Yaskawa INFORM job: X2_27-28(-50,-90).JBI

/JOB
//NAME X2_27-28(-50,-90)
//POS
///NPOS 347,347,347,16,0,0
///TOOL 0
///POSTYPE PULSE
///PULSE
C00000=2348,-136985,-121477,16,96092,119
C00001=-102627,-116827,-115343,-23688,103226,44542
C00002=-115004,-86962,-92134,-24001,100691,40453
C00003=-118842,-87386,-89376,-23795,97842,39618
C00004=-120381,-87384,-88200,-23717,96741,39273
C00005=-120377,-87274,-86494,-23659,95829,39457
C00006=-120358,-87289,-86697,-23665,95942,39442
C00007=-122537,-87238,-86673,-23616,95334,38762
C00008=-120358,-87289,-86697,-23665,95942,39442
C00009=-120413,-87366,-86683,-23662,95882,39433
C00010=-120414,-83407,-84990,-23721,96794,39250
C00011=-120413,-87366,-86683,-23662,95882,39433
C00012=-118874,-87417,-87880,-23731,96972,39781
C00013=-115033,-87126,-90695,-23913,99792,40627
C00014=-115188,-84882,-91157,-24044,101067,40307
C00015=-118973,-85347,-88418,-23826,98226,39491
C00016=-120455,-85363,-87251,-23745,97137,39166
C00017=-120452,-85286,-85558,-23683,96217,39352
C00018=-120487,-85295,-85812,-23691,96347,39313
C00019=-122635,-85238,-85785,-23639,95749,38643
C00020=-120487,-85295,-85812,-23691,96347,39313
C00021=-120483,-89746,-89095,-23675,96102,39363
C00022=-120398,-93403,-88367,-23560,93986,39817
C00023=-120400,-89378,-86736,-23609,94965,39621
C00024=-120398,-93403,-88367,-23560,93986,39817
C00025=-114754,-95185,-95401,-23812,98729,40947
C00026=-113817,-96176,-94667,-23309,84492,38861
C00027=-117813,-93582,-90807,-22657,82424,37804
C00028=-119373,-92438,-89214,-22393,81636,37384
C00029=-121634,-92435,-89210,-21971,81030,36673
C00030=-120812,-92629,-89389,-22126,81259,36930
C00031=-120809,-92377,-87626,-22175,80372,37096
C00032=-120812,-92629,-89389,-22126,81259,36930
C00033=-120909,-77641,-83091,-21971,84792,36245
C00034=-120897,-73822,-81314,-21956,85603,36101
C00035=-120909,-77641,-83091,-21971,84792,36245
C00036=-115943,-80689,-88441,-22878,87717,37472
C00037=-114304,-84462,-91699,-24296,79100,50020
C00038=-117993,-82622,-88033,-23316,76858,49124
C00039=-119438,-81769,-86512,-22922,76000,48762
C00040=-121534,-81768,-86509,-22277,75434,48100
C00041=-120893,-81605,-86471,-22471,75662,48293
C00042=-120882,-79116,-84088,-22491,75491,48329
C00043=-120893,-81605,-86471,-22471,75662,48293
C00044=-120874,-97072,-87829,-23296,69089,49605
C00045=-120882,-99825,-87797,-23508,67765,49878
C00046=-120874,-97072,-87829,-23296,69089,49605
C00047=-115137,-101258,-93439,-24799,71949,51221
C00048=-121122,-106374,-107449,1374,89824,2285
C00049=-126924,-83388,-91593,24529,79629,-49999
C00050=-123244,-81641,-87969,23551,77363,-49118
C00051=-121801,-80822,-86464,23159,76497,-48761
C00052=-119718,-80838,-86473,22519,75929,-48107
C00053=-120355,-80669,-86431,22711,76157,-48297
C00054=-120355,-78205,-84050,22728,75972,-48332
C00055=-120355,-80669,-86431,22711,76157,-48297
C00056=-120389,-96242,-87887,23521,69604,-49623
C00057=-120385,-99021,-87874,23730,68282,-49899
C00058=-120389,-96242,-87887,23521,69604,-49623
C00059=-126112,-100299,-93445,25011,72503,-51215
C00060=-127424,-95125,-94496,23537,84985,-38865
C00061=-123439,-92623,-90674,22887,82890,-37821
C00062=-121881,-91514,-89094,22623,82092,-37406
C00063=-119636,-91530,-89104,22205,81483,-36703
C00064=-120453,-91715,-89278,22359,81714,-36957
C00065=-120449,-91492,-87527,22405,80819,-37124
C00066=-120453,-91715,-89278,22359,81714,-36957
C00067=-120324,-76745,-82936,22209,85198,-36262
C00068=-120328,-72933,-81149,22194,85997,-36116
C00069=-120324,-76745,-82936,22209,85198,-36262
C00070=-125282,-79685,-88237,23118,88153,-37475
C00071=-126053,-84105,-90945,24270,101400,-40334
C00072=-121317,-84665,-86997,23961,97551,-39378
C00073=-120794,-84655,-86302,23916,97014,-39294
C00074=-120791,-84616,-85408,23898,96528,-39392
C00075=-120757,-84623,-85661,23907,96658,-39353
C00076=-118619,-84583,-85646,23856,96058,-38687
C00077=-120757,-84623,-85661,23907,96658,-39353
C00078=-120851,-89642,-89189,23884,96311,-39457
C00079=-120861,-92728,-88235,23770,94318,-39863
C00080=-120850,-88708,-86596,23821,95285,-39665
C00081=-120861,-92728,-88235,23770,94318,-39863
C00082=-126087,-84100,-90943,24271,101411,-40344
C00083=-126241,-86175,-91925,24226,101032,-40481
C00084=-121422,-86671,-87791,23936,97086,-39512
C00085=-120872,-86641,-86990,23895,96491,-39430
C00086=-120871,-86598,-86346,23873,96146,-39499
C00087=-120890,-86611,-86548,23880,96260,-39483
C00088=-118722,-86577,-86536,23832,95649,-38808
C00089=-120890,-86611,-86548,23880,96260,-39483
C00090=-105063,-136064,-103329,13656,63018,-16453
C00091=-105943,-129413,-101511,13642,65401,-16501
C00092=-120836,-86689,-86535,23876,96200,-39475
C00093=-126205,-86358,-90494,24135,100129,-40655
C00094=-125851,-82973,-83923,27955,66645,-49280
C00095=-122078,-79433,-79887,26568,64829,-48204
C00096=-120742,-75548,-77663,25886,64978,-47626
C00097=-120603,-87757,-78081,27201,59519,-48941
C00098=-120577,-18765,-47570,25588,110640,-38043
C00099=-109277,-31294,-61129,11102,108845,-34159
C00100=-108190,-73941,-84391,11784,95620,-26863
C00101=-120412,-77832,-82211,23564,93525,-30308
C00102=-120295,-129804,-92806,30270,50820,-51385
C00103=-120103,-142543,-87811,36899,40276,-55620
C00104=-123719,-144899,-89705,38330,41729,-57027
C00105=-131684,-150990,-93667,41315,44633,-60156
C00106=-129569,-143343,-101170,37382,56065,-55166
C00107=-120626,-84262,-98768,23738,98439,-36527
C00108=-120626,-85138,-96217,23600,96582,-36901
C00109=-120626,-85402,-95162,23554,95859,-37045
C00110=-120626,-85402,-95166,23554,95862,-37044
C00111=-120625,-86138,-87819,24831,69352,-42364
C00112=-120624,-85351,-79999,28656,54651,-46082
C00113=-120624,-83851,-73296,29505,52526,-46737
C00114=-120624,-85502,-80901,24858,69157,-42411
C00115=-120625,-86091,-86368,23338,89997,-38197
C00116=-120623,-90747,-88263,23328,88867,-38416
C00117=-120625,-86141,-87502,23348,90617,-38076
C00118=-120625,-86117,-90396,23390,92270,-37753
C00119=-121122,-106374,-107449,1374,89824,2285
C00120=-115389,-83619,-83840,-27729,66202,49282
C00121=-119161,-80016,-79774,-26335,64406,48194
C00122=-120089,-78340,-77954,-26002,63882,47941
C00123=-118763,-53285,-67852,-25424,88543,43198
C00124=-120520,-20811,-48856,-25337,110383,38072
C00125=-120672,-56250,-71200,-24620,106276,38936
C00126=-122381,-110474,-92211,-22628,69435,43351
C00127=-117850,-143004,-85318,-49461,33775,58563
C00128=-117015,-147748,-80398,-56682,30834,62523
C00129=-116407,-166632,-89102,-63406,28902,66105
C00130=-115676,-54235,-75024,-25023,110799,39825
C00131=-118805,-64147,-80292,-27733,101935,40879
C00132=-120626,-85310,-99014,-23481,98015,36524
C00133=-120626,-86187,-96453,-23350,96148,36894
C00134=-120946,-86934,-95392,-23260,95104,36986
C00135=-120769,-87776,-95791,-23270,94982,37074
C00136=-120625,-87052,-87833,-24600,68847,42365
C00137=-120546,-85594,-79665,-28457,54282,46089
C00138=-120538,-84322,-72984,-29356,52066,46772
C00139=-120625,-86297,-80888,-24632,68687,42397
C00140=-119608,-72473,-79941,-24560,98029,43290
C00141=-120361,-60134,-73697,-25010,105724,48535
C00142=-120625,-87037,-87669,-23119,90208,38053
C00143=-120626,-87011,-90570,-23155,91868,37731
C00144=-120666,-77011,-108669,-24508,106824,34682
C00145=-69969,-70044,-127853,26190,66176,-42607
C00146=-164066,-57873,-122395,24689,68505,-41679
C00147=-164066,-57873,-122395,24689,68505,-41679
C00148=-160176,-49519,-119791,24551,119921,-39872
C00149=-160176,-63483,-121326,22850,113002,-41438
C00150=-158640,-65340,-120741,22195,111473,-41297
C00151=-158591,-68589,-120293,21868,109653,-41643
C00152=-157443,-69457,-121106,21570,109470,-41332
C00153=-156525,-70687,-121652,21280,109008,-41144
C00154=-157421,-68776,-121134,21620,109807,-41260
C00155=-165312,-86424,-128504,22962,107296,-44197
C00156=-165830,-86354,-127308,22986,106767,-44469
C00157=-165199,-83493,-126223,22948,107364,-44147
C00158=-166594,-89849,-128602,23030,106020,-44865
C00159=-164066,-57873,-122395,24689,117052,-41679
C00160=-137183,-48540,-113103,27062,110870,-33097
C00161=-133437,-50146,-110771,25387,107987,-32705
C00162=-131981,-50551,-109735,24766,106894,-32528
C00163=-131972,-53362,-109280,24521,105318,-32870
C00164=-131636,-52132,-109559,24518,105977,-32629
C00165=-130703,-53161,-109590,24138,105304,-32500
C00166=-129879,-53398,-109717,23857,105082,-32305
C00167=-131928,-52773,-109383,24556,105642,-32786
C00168=-129764,-110950,-131053,20350,81074,-33499
C00169=-129689,-122862,-131886,20674,75787,-34382
C00170=-129370,-114001,-129067,20345,78360,-33827
C00171=-129689,-122862,-131886,20674,75787,-34382
C00172=-132778,-100905,-131254,21387,86712,-33498
C00173=-143318,-75184,-130722,7426,108145,-5953
C00174=-142042,-70835,-125479,6985,107076,-5675
C00175=-141569,-69161,-123389,6821,106623,-5573
C00176=-141558,-72780,-123049,6738,104567,-5686
C00177=-141593,-72294,-123187,6761,104902,-5677
C00178=-140967,-66354,-120569,6623,106293,-5428
C00179=-141593,-72294,-123187,6761,104902,-5677
C00180=-143345,-79213,-130741,7340,106105,-6087
C00181=-143299,-74412,-130544,7434,108429,-5930
C00182=-142026,-70178,-125329,6991,107319,-5656
C00183=-141554,-68541,-123249,6826,106852,-5556
C00184=-141544,-72173,-122918,6742,104795,-5669
C00185=-141535,-71558,-123086,6755,105212,-5644
C00186=-140912,-65651,-120469,6618,106588,-5397
C00187=-141535,-71558,-123086,6755,105212,-5644
C00188=-143280,-78289,-130595,7337,106482,-6046
C00189=-143232,-73654,-130370,7428,108704,-5895
C00190=-141965,-69530,-125182,6983,107555,-5626
C00191=-141496,-67928,-123110,6817,107076,-5527
C00192=-141485,-71574,-122787,6732,105017,-5641
C00193=-141522,-70879,-122980,6762,105492,-5624
C00194=-140900,-65004,-120364,6625,106853,-5379
C00195=-141522,-70879,-122980,6762,105492,-5624
C00196=-143263,-77436,-130447,7347,106826,-6020
C00197=-97122,-37708,-107994,-29413,114613,34215
C00198=-100765,-40257,-106178,-27624,111617,33971
C00199=-102190,-41052,-105346,-26964,110463,33848
C00200=-102184,-43828,-104954,-26656,108968,34218
C00201=-102229,-43254,-105047,-26705,109274,34130
C00202=-104151,-44223,-105589,-26045,108681,33706
C00203=-102229,-43254,-105047,-26705,109274,34130
C00204=-102390,-95092,-126215,-23236,87986,35228
C00205=-102126,-106454,-127212,-23433,83236,36243
C00206=-102723,-99043,-124596,-23148,85111,35678
C00207=-102126,-106454,-127212,-23433,83236,36243
C00208=-98351,-76946,-122874,-24964,95636,34932
C00209=-98001,-57475,-123101,-17996,113820,36592
C00210=-101536,-60773,-120906,-16470,110382,36160
C00211=-102910,-63141,-119733,-15828,108317,36071
C00212=-102916,-65026,-119479,-15713,107233,36217
C00213=-102928,-64308,-119579,-15751,107645,36158
C00214=-105169,-65555,-120144,-15037,107042,35610
C00215=-102928,-64308,-119579,-15751,107645,36158
C00216=-100368,-93898,-131351,-15864,100368,37874
C00217=-97661,-87630,-128580,-16731,102276,38427
C00218=-97996,-84252,-127310,-16710,103135,38207
C00219=-97637,-87591,-128732,-16747,102389,38418
C00220=-98001,-57475,-123101,-17996,113820,36592
C00221=-99672,-7498,-88471,-25376,120102,35641
C00222=-102088,-13346,-89114,-23936,117260,35660
C00223=-103047,-14853,-89113,-23458,116364,35598
C00224=-103070,-15280,-89318,-23419,116275,35613
C00225=-103053,-14956,-89343,-23464,116445,35580
C00226=-111428,-26181,-98637,-10737,112296,30408
C00227=-102060,-12538,-89166,-24052,117675,35572
C00228=-99645,-6651,-88487,-25511,120511,35544
C00229=-110953,-13508,-91662,-10573,109125,-24437
C00230=-110055,-18058,-91129,-10746,106581,-23991
C00231=-118115,-24092,-94041,1176,104714,-22608
C00232=-109847,-18561,-90498,-10785,105963,-23883
C00233=-111445,-19708,-91242,-10156,105696,-24257
C00234=-118682,-20843,-91970,-7294,105023,-25985
C00235=-108853,-8664,-84384,-24098,112429,-23291
C00236=-120831,-18883,-92219,-6481,106051,-26563
C00237=-108247,-47697,-110693,-11257,103619,-23266
C00238=-108001,-45758,-107370,-11293,102615,-23108
C00239=-93743,-22704,-93084,-31932,116237,-9910
C00240=-103043,-28379,-96833,-28832,113378,-11880
C00241=-99567,-22662,-96038,-30605,116358,-11712
C00242=-121744,-14004,-92551,-6221,108699,-26920
C00243=-120102,-53038,-115079,8947,92663,-44391
C00244=-120610,-122376,-128753,45788,73253,-81068
C00245=-120610,-123649,-126232,46257,71693,-81820
C00246=-114032,-121391,-128573,37709,71856,-79804
C00247=-110037,-117352,-129528,31885,73379,-77591
C00248=-111712,-119204,-129441,32400,72227,-78861
C00249=-111738,-118516,-129193,32380,72408,-78818
C00250=-117085,-123222,-129338,33957,68924,-83144
C00251=-117209,-115215,-126517,33557,70967,-82546
C00252=-120611,-120126,-130997,36594,78100,-80978
C00253=-120611,-116611,-133297,36284,80720,-80097
C00254=-120611,-116611,-133297,36284,54343,-80097
C00255=-99428,-107843,-133398,-6584,68498,-81557
C00256=-78879,-54177,-103402,-55937,89044,-85268
C00257=-78429,-99723,-127104,-45672,96643,-84222
C00258=-82364,-110385,-127773,-44232,91185,-83459
C00259=-84004,-114197,-127845,-43759,89024,-83232
C00260=-84284,-115490,-128627,-43147,88793,-83830
C00261=-84701,-116384,-128576,-43135,87361,-83811
C00262=-93522,-101978,-128819,-33845,95617,-84197
C00263=-94093,-97143,-127093,-33800,96609,-84705
C00264=-92227,-97102,-128188,-34391,97842,-84417
C00265=-83296,-105916,-131418,-40048,95342,-83077
C00266=-112976,-81346,-133029,-11053,104292,-84731
C00267=-138914,-76030,-130615,14013,102422,-84743
C00268=-139405,-82424,-128484,14961,97637,-85019
C00269=-139021,-85906,-128645,14753,95944,-85117
C00270=-122175,-93047,-130840,-6754,91446,-83840
C00271=-120351,-90450,-129884,-7457,92320,-83370
C00272=-122216,-90116,-129760,-6745,92278,-83897
C00273=-121098,-81728,-131688,-7259,97815,-83901
C00274=-117564,-73996,-132555,-6245,103794,-67045
C00275=-120619,-75058,-128623,5257,106122,-114
C00276=-120619,-82255,-128190,5150,102172,-284
C00277=-120619,-84669,-127718,5117,100646,-349
C00278=-112025,-83330,-127195,2462,100682,2074
C00279=-125417,-84542,-127836,6591,101068,-1686
C00280=-115735,-84377,-127810,3614,100638,1033
C00281=-120619,-81538,-128040,5156,102448,-272
C00282=-120619,-74311,-128456,5266,106402,-102
C00283=-120619,-74726,-128566,-4732,106271,192
C00284=-120619,-81960,-128145,-4635,102308,346
C00285=-120619,-85178,-127943,-4602,100537,414
C00286=-130218,-83751,-127399,-1640,100634,-2293
C00287=-124486,-85286,-127816,-3408,100245,-674
C00288=-123475,-85288,-127855,-3720,100302,-390
C00289=-120619,-82679,-128294,-4629,102031,356
C00290=-132569,-75475,-129249,-4725,105990,203
C00291=-136339,-73848,-128583,-3524,106271,-812
C00292=-115610,-90997,-132796,-9664,98154,-47330
C00293=-101030,-93647,-129382,-39129,95529,-59479
C00294=-126122,-118259,-133558,-37742,75798,-85079
C00295=-126123,-123502,-128947,-38676,71399,-83468
C00296=-125878,-125726,-128593,-39051,70435,-82992
C00297=-125899,-125877,-129038,-38326,70614,-83857
C00298=-125755,-123018,-128156,-38195,71411,-84090
C00299=-123565,-128869,-131754,-35345,71844,-80466
C00300=-127099,-118299,-127920,-31029,69914,-80741
C00301=-124670,-119490,-131862,-32313,77272,-81796
C00302=-123468,-105545,-131306,-32649,85926,-83785
C00303=-123468,-105545,-131306,-32649,65045,-83785
C00304=-137523,-77632,-116284,43410,62933,-71250
C00305=-137523,-77632,-116284,43410,93706,-71250
C00306=-133557,-83369,-115610,41847,89536,-71423
C00307=-133747,-120555,-122786,46504,70292,-79425
C00308=-131929,-100191,-119235,41912,80202,-73781
C00309=-130616,-80903,-112666,40052,87263,-70292
C00310=-128915,-78749,-114170,37546,91382,-70207
C00311=-127369,-79400,-118715,34661,97087,-70456
C00312=-130909,-72948,-119538,36294,101438,-70254
C00313=-103939,-76664,-132684,5369,102917,-72052
C00314=-89328,-90531,-135287,-12506,96574,-73027
C00315=-80068,-79251,-126452,-22073,101797,-73002
C00316=-79731,-82396,-126595,-22049,100450,-72647
C00317=-79925,-81438,-126213,-22008,100648,-72742
C00318=-98451,-112019,-134925,6092,80988,-72427
C00319=-96878,-106433,-133907,2900,84129,-72442
C00320=-94333,-103386,-132879,1852,84995,-71667
C00321=-89270,-85342,-132616,-4377,96009,-71566
C00322=-120927,-40602,-113932,15942,113021,-53571
C00323=-134131,-13261,-91828,23304,117904,-34003
C00324=-134130,-17922,-91482,22725,115495,-34532
C00325=-134178,-18161,-90930,22645,115075,-34636
C00326=-134130,-19018,-91366,22584,114907,-34660
C00327=-134135,-19080,-91406,22584,114899,-34666
C00328=-130040,-16797,-91734,17058,116519,-30349
C00329=-134130,-17121,-91555,22821,115917,-34441
C00330=-134485,-13609,-94717,23816,119438,-33744
C00331=-134125,-15266,-91655,12564,108610,23590
C00332=-134126,-19967,-91222,12356,105989,23311
C00333=-128619,-18785,-91351,4606,108870,22773
C00334=-134001,-21196,-91423,12272,105476,23287
C00335=-133837,-21232,-91027,12191,105205,23306
C00336=-133810,-21099,-91074,12188,105299,23320
C00337=-142675,1303,-75956,28153,117136,18516
C00338=-136270,-18169,-92488,13326,107877,22987
C00339=-160414,-17591,-92076,34517,119430,9586
C00340=-156591,-5353,-82577,31368,124461,10572
C00341=-145789,-11555,-87834,25790,123238,6673
C00342=-150771,-16897,-91755,28044,119951,5168
C00343=-137962,-9823,-90715,14308,111174,22977
C00344=-134122,-37576,-106581,14512,53534,24067
C00345=-90631,-69256,-111328,9893,26432,16435
C00346=2348,-136985,-121477,16,96092,119
BC00000=133260,671337,1075175
BC00001=133260,816101,1075175
BC00002=133260,816101,1075175
BC00003=133260,816101,1075175
BC00004=133260,816101,1075175
BC00005=133260,816101,1075175
BC00006=133260,816101,1075175
BC00007=133260,816101,1075175
BC00008=133260,816101,1075175
BC00009=133260,816101,1075175
BC00010=133260,816101,1075175
BC00011=133260,816101,1075175
BC00012=133260,816101,1075175
BC00013=133260,816101,1075175
BC00014=133352,784558,1075175
BC00015=133352,784558,1075175
BC00016=133352,784558,1075175
BC00017=133352,784558,1075175
BC00018=133352,784558,1075175
BC00019=133352,784558,1075175
BC00020=133352,784558,1075175
BC00021=133352,784558,1075175
BC00022=133352,784558,1075175
BC00023=133352,784558,1075175
BC00024=133352,784558,1075175
BC00025=133352,784558,1075175
BC00026=104493,781490,1075175
BC00027=104493,781490,1075175
BC00028=104493,781490,1075175
BC00029=104493,781490,1075175
BC00030=104493,781490,1075175
BC00031=104493,781490,1075175
BC00032=104493,781490,1075175
BC00033=104493,781490,1075175
BC00034=104493,781490,1075175
BC00035=104493,781490,1075175
BC00036=104493,781490,1075175
BC00037=104598,779058,1075175
BC00038=104598,779058,1075175
BC00039=104598,779058,1075175
BC00040=104598,779058,1075175
BC00041=104598,779058,1075175
BC00042=104598,779058,1075175
BC00043=104598,779058,1075175
BC00044=104598,779058,1075175
BC00045=104598,779058,1075175
BC00046=104598,779058,1075175
BC00047=104598,779058,1075175
BC00048=209921,798961,1075175
BC00049=330511,779036,1075175
BC00050=330511,779036,1075175
BC00051=330511,779036,1075175
BC00052=330511,779036,1075175
BC00053=330511,779036,1075175
BC00054=330511,779036,1075175
BC00055=330511,779036,1075175
BC00056=330511,779036,1075175
BC00057=330511,779036,1075175
BC00058=330511,779036,1075175
BC00059=330511,779036,1075175
BC00060=330352,781550,1075175
BC00061=330352,781550,1075175
BC00062=330352,781550,1075175
BC00063=330352,781550,1075175
BC00064=330352,781550,1075175
BC00065=330352,781550,1075175
BC00066=330352,781550,1075175
BC00067=330352,781550,1075175
BC00068=330352,781550,1075175
BC00069=330352,781550,1075175
BC00070=330352,781550,1075175
BC00071=301652,784810,1075175
BC00072=301653,784809,1075174
BC00073=301653,784809,1075173
BC00074=301652,784810,1075175
BC00075=301652,784810,1075175
BC00076=301652,784810,1075175
BC00077=301652,784810,1075175
BC00078=301652,784810,1075175
BC00079=301652,784810,1075175
BC00080=301652,784810,1075175
BC00081=301652,784810,1075175
BC00082=301652,784810,1075175
BC00083=301940,816351,1075175
BC00084=301940,816351,1075175
BC00085=301940,816351,1075175
BC00086=301940,816351,1075175
BC00087=301940,816351,1075175
BC00088=301940,816351,1075175
BC00089=301940,816351,1075175
BC00090=301940,816351,1075175
BC00091=301940,816351,1075175
BC00092=301940,816351,1075175
BC00093=301940,816351,1075175
BC00094=304921,767834,1075175
BC00095=304921,767834,1075175
BC00096=304921,767834,1075175
BC00097=304921,767834,1075175
BC00098=304921,767834,1075175
BC00099=304921,767834,1075175
BC00100=304921,767834,1075175
BC00101=304921,767834,1075175
BC00102=304921,767834,1075175
BC00103=304921,767834,1075175
BC00104=304921,767834,1075175
BC00105=304921,767834,1075175
BC00106=308198,778885,1075186
BC00107=321964,825300,1075229
BC00108=327565,826190,1075229
BC00109=329805,826547,1075229
BC00110=329800,825010,1075229
BC00111=329695,783757,1075229
BC00112=329661,765313,1075229
BC00113=329637,751680,1075229
BC00114=329672,769766,1075229
BC00115=329747,798928,1075229
BC00116=329696,782419,1075229
BC00117=327455,782039,1075229
BC00118=321854,781091,1075229
BC00119=209921,798961,1075175
BC00120=130067,767697,1075175
BC00121=130067,767697,1075175
BC00122=130067,767697,1075175
BC00123=130067,767697,1075175
BC00124=130067,767697,1075175
BC00125=130067,767697,1075175
BC00126=130067,767697,1075175
BC00127=130067,767697,1075175
BC00128=130067,767697,1075175
BC00129=130067,767697,1075175
BC00130=130067,767697,1075175
BC00131=129391,769992,1075177
BC00132=113149,825170,1075229
BC00133=107572,826093,1075229
BC00134=105340,826462,1075229
BC00135=105336,824926,1075229
BC00136=105231,783763,1075229
BC00137=105197,765408,1075229
BC00138=105173,751768,1075229
BC00139=105208,769749,1075229
BC00140=105282,798844,1075229
BC00141=105231,782335,1075229
BC00142=107462,781943,1075229
BC00143=113040,780963,1075229
BC00144=113040,780963,1075229
BC00145=61101,668037,1075175
BC00146=61101,668037,1075175
BC00147=61101,845904,1075175
BC00148=61101,845904,1072970
BC00149=61101,845904,1075175
BC00150=61101,845904,1075175
BC00151=61101,845904,1075175
BC00152=61101,845904,1075175
BC00153=61101,845904,1075175
BC00154=61101,845904,1075175
BC00155=61101,845904,1075175
BC00156=61101,845904,1075175
BC00157=61101,845904,1075175
BC00158=61101,845904,1075175
BC00159=61101,845904,1075175
BC00160=23296,842661,1075175
BC00161=23296,842661,1075175
BC00162=23296,842661,1075175
BC00163=23296,842661,1075175
BC00164=23296,842661,1075175
BC00165=23296,842661,1075175
BC00166=23296,842661,1075175
BC00167=23296,842661,1075175
BC00168=23296,842661,1075175
BC00169=23296,842661,1075175
BC00170=23296,842661,1075175
BC00171=23296,842661,1075175
BC00172=23296,842661,1075175
BC00173=188993,843499,1075175
BC00174=188993,843499,1075175
BC00175=188993,843499,1075175
BC00176=188993,843499,1075175
BC00177=188993,843499,1075175
BC00178=188993,843499,1075175
BC00179=188993,843499,1075175
BC00180=188993,843499,1075175
BC00181=244510,843369,1075175
BC00182=244510,843369,1075175
BC00183=244510,843369,1075175
BC00184=244510,843369,1075175
BC00185=244510,843369,1075175
BC00186=244510,843369,1075175
BC00187=244510,843369,1075175
BC00188=244510,843369,1075175
BC00189=299392,843255,1075175
BC00190=299392,843255,1075175
BC00191=299392,843255,1075175
BC00192=299392,843255,1075175
BC00193=299392,843255,1075175
BC00194=299392,843255,1075175
BC00195=299392,843255,1075175
BC00196=299392,843255,1075175
BC00197=398174,838715,1075175
BC00198=398174,838715,1075175
BC00199=398174,838715,1075175
BC00200=398174,838715,1075175
BC00201=398174,838715,1075175
BC00202=398174,838715,1075175
BC00203=398174,838715,1075175
BC00204=398174,838715,1075175
BC00205=398174,838715,1075175
BC00206=398174,838715,1075175
BC00207=398174,838715,1075175
BC00208=398174,838715,1075175
BC00209=398174,834777,1075175
BC00210=398174,834777,1075175
BC00211=398174,834777,1075175
BC00212=398174,834777,1075175
BC00213=398174,834777,1075175
BC00214=398174,834777,1075175
BC00215=398174,834777,1075175
BC00216=398174,834777,1075175
BC00217=398174,834777,1075175
BC00218=398174,834777,1075175
BC00219=398174,834777,1075175
BC00220=398174,834777,1075175
BC00221=398174,789787,1075175
BC00222=398174,792647,1075175
BC00223=398174,793791,1075175
BC00224=398174,798395,1075175
BC00225=398174,812684,1075175
BC00226=398174,817289,1075175
BC00227=398174,816145,1075175
BC00228=398174,813286,1075175
BC00229=398174,772020,1075175
BC00230=398174,777054,1075175
BC00231=398174,779068,1075175
BC00232=398174,779068,1075175
BC00233=398174,782408,1075175
BC00234=398174,796035,1075175
BC00235=398173,799310,1075174
BC00236=398174,797352,1075175
BC00237=398174,797352,1075175
BC00238=398174,797352,1075175
BC00239=398174,797352,1075175
BC00240=398174,797352,1075175
BC00241=398174,797352,1075175
BC00242=398174,792318,1075175
BC00243=368052,813684,1075175
BC00244=305396,862056,1075175
BC00245=311030,862741,1075175
BC00246=313284,863016,1075175
BC00247=314036,883858,1075171
BC00248=316331,884912,1075171
BC00249=316331,884912,1075171
BC00250=325372,889063,1075173
BC00251=325372,889063,1075173
BC00252=323920,889033,1075175
BC00253=319279,888490,1075175
BC00254=319279,888490,1075175
BC00255=354646,872242,1075175
BC00256=398174,845986,1075175
BC00257=398174,861280,1075175
BC00258=398174,861992,1075175
BC00259=398174,862277,1075175
BC00260=398174,883807,1075175
BC00261=398174,882455,1075175
BC00262=398174,890246,1075175
BC00263=398174,890246,1075175
BC00264=398174,890259,1075175
BC00265=398174,890291,1075175
BC00266=398174,883515,1075175
BC00267=398174,877168,1075175
BC00268=398174,877782,1075175
BC00269=398174,878199,1075175
BC00270=398174,878161,1075175
BC00271=398174,878161,1075175
BC00272=398174,878161,1075175
BC00273=398174,877847,1075175
BC00274=361291,866796,1075175
BC00275=206073,840782,1075175
BC00276=206803,846220,1075175
BC00277=207094,848395,1075175
BC00278=207094,848395,1075175
BC00279=265264,848258,1075175
BC00280=265264,848258,1075175
BC00281=264972,846083,1075175
BC00282=264242,840645,1075175
BC00283=226811,840688,1075175
BC00284=226153,846129,1075175
BC00285=225889,848305,1075175
BC00286=225889,848305,1075175
BC00287=182410,848408,1075175
BC00288=167720,848443,1075175
BC00289=167983,846266,1075175
BC00290=168641,840825,1075175
BC00291=168641,840825,1075175
BC00292=110843,840825,1075175
BC00293=117034,848211,1075175
BC00294=129099,862603,1075175
BC00295=123513,863314,1075175
BC00296=121279,863599,1075175
BC00297=120610,884955,1075175
BC00298=120610,884955,1075175
BC00299=111851,888645,1075175
BC00300=111851,888642,1075173
BC00301=111110,889324,1075174
BC00302=115335,889093,1075175
BC00303=115335,889093,1075175
BC00304=15,847247,1075175
BC00305=15,847247,1075175
BC00306=15,847933,1075175
BC00307=15,848207,1075175
BC00308=15,869372,1075175
BC00309=15,867972,1075175
BC00310=15,874442,1075175
BC00311=15,883049,1075175
BC00312=15,883104,1075175
BC00313=5550,880629,1075175
BC00314=11084,884590,1075175
BC00315=10009,885638,1075175
BC00316=9623,886015,1075175
BC00317=9623,886015,1075175
BC00318=15,886096,1075175
BC00319=15,885980,1075175
BC00320=15,885980,1075175
BC00321=15,885783,1075175
BC00322=5547,839492,1075175
BC00323=20493,791516,1075175
BC00324=25334,794353,1075175
BC00325=27270,795487,1075175
BC00326=27300,800091,1075175
BC00327=27334,814381,1075175
BC00328=27329,817326,1075175
BC00329=25390,817851,1075175
BC00330=20549,815014,1075175
BC00331=41925,772454,1075175
BC00332=40308,777496,1075175
BC00333=39661,779513,1075175
BC00334=39661,779513,1075175
BC00335=42967,782837,1075175
BC00336=56491,796400,1075175
BC00337=56491,796400,1075175
BC00338=60452,797699,1075175
BC00339=60452,797699,1075175
BC00340=60451,797698,1075172
BC00341=60451,797698,1075172
BC00342=60451,797698,1075172
BC00343=62069,792657,1075175
BC00344=62069,792657,1075175
BC00345=84756,753994,1075175
BC00346=133260,671337,1075175
EC00000=-443420,-556475
EC00001=-443420,-556475
EC00002=-443420,-556475
EC00003=-443420,-556475
EC00004=-443420,-556475
EC00005=-443420,-556475
EC00006=-443420,-556475
EC00007=-443420,-556475
EC00008=-443420,-556475
EC00009=-443420,-556475
EC00010=-443420,-556475
EC00011=-443420,-556475
EC00012=-443420,-556475
EC00013=-443420,-556475
EC00014=-443420,-556475
EC00015=-443420,-556475
EC00016=-443420,-556475
EC00017=-443420,-556475
EC00018=-443420,-556475
EC00019=-443420,-556475
EC00020=-443420,-556475
EC00021=-443420,-556475
EC00022=-443420,-556475
EC00023=-443420,-556475
EC00024=-443420,-556475
EC00025=-443420,-556475
EC00026=-443420,-556475
EC00027=-443420,-556475
EC00028=-443420,-556475
EC00029=-443420,-556475
EC00030=-443420,-556475
EC00031=-443420,-556475
EC00032=-443420,-556475
EC00033=-443420,-556475
EC00034=-443420,-556475
EC00035=-443420,-556475
EC00036=-443420,-556475
EC00037=-443420,-556475
EC00038=-443420,-556475
EC00039=-443420,-556475
EC00040=-443420,-556475
EC00041=-443420,-556475
EC00042=-443420,-556475
EC00043=-443420,-556475
EC00044=-443420,-556475
EC00045=-443420,-556475
EC00046=-443420,-556475
EC00047=-443420,-556475
EC00048=-443420,-556475
EC00049=-443420,-556475
EC00050=-443420,-556475
EC00051=-443420,-556475
EC00052=-443420,-556475
EC00053=-443420,-556475
EC00054=-443420,-556475
EC00055=-443420,-556475
EC00056=-443420,-556475
EC00057=-443420,-556475
EC00058=-443420,-556475
EC00059=-443420,-556475
EC00060=-443420,-556475
EC00061=-443420,-556475
EC00062=-443420,-556475
EC00063=-443420,-556475
EC00064=-443420,-556475
EC00065=-443420,-556475
EC00066=-443420,-556475
EC00067=-443420,-556475
EC00068=-443420,-556475
EC00069=-443420,-556475
EC00070=-443420,-556475
EC00071=-443420,-556475
EC00072=-443419,-556476
EC00073=-443418,-556476
EC00074=-443420,-556475
EC00075=-443420,-556475
EC00076=-443420,-556475
EC00077=-443420,-556475
EC00078=-443420,-556475
EC00079=-443420,-556475
EC00080=-443420,-556475
EC00081=-443420,-556475
EC00082=-443420,-556475
EC00083=-443420,-556475
EC00084=-443420,-556475
EC00085=-443420,-556475
EC00086=-443420,-556475
EC00087=-443420,-556475
EC00088=-443420,-556475
EC00089=-443420,-556475
EC00090=-443420,-556475
EC00091=-443420,-556475
EC00092=-443420,-556475
EC00093=-443420,-556475
EC00094=-443420,-556475
EC00095=-443420,-556475
EC00096=-443420,-556475
EC00097=-443420,-556475
EC00098=-443420,-556475
EC00099=-443420,-556475
EC00100=-443420,-556475
EC00101=-443420,-556475
EC00102=-443420,-556475
EC00103=-443420,-556475
EC00104=-443420,-556475
EC00105=-443420,-556475
EC00106=-443420,-556475
EC00107=-443420,-556475
EC00108=-443420,-556475
EC00109=-443420,-556475
EC00110=-443420,-556475
EC00111=-443420,-556475
EC00112=-443420,-556475
EC00113=-443420,-556475
EC00114=-443420,-556475
EC00115=-443420,-556475
EC00116=-443420,-556475
EC00117=-443420,-556475
EC00118=-443420,-556475
EC00119=-443420,-556475
EC00120=-443420,-556475
EC00121=-443420,-556475
EC00122=-443420,-556475
EC00123=-443420,-556475
EC00124=-443420,-556475
EC00125=-443420,-556475
EC00126=-443420,-556475
EC00127=-443420,-556475
EC00128=-443420,-556475
EC00129=-443420,-556475
EC00130=-443420,-556475
EC00131=-443420,-556475
EC00132=-443420,-556475
EC00133=-443420,-556475
EC00134=-443420,-556475
EC00135=-443420,-556475
EC00136=-443420,-556475
EC00137=-443420,-556475
EC00138=-443420,-556475
EC00139=-443420,-556475
EC00140=-443420,-556475
EC00141=-443420,-556475
EC00142=-443420,-556475
EC00143=-443420,-556475
EC00144=-443420,-556475
EC00145=-798156,-556475
EC00146=-798156,-556475
EC00147=-798156,-556475
EC00148=-798156,-556475
EC00149=-798156,-556475
EC00150=-798156,-556475
EC00151=-798156,-556475
EC00152=-798156,-556475
EC00153=-798156,-556475
EC00154=-798156,-556475
EC00155=-798156,-556475
EC00156=-798156,-556475
EC00157=-798156,-556475
EC00158=-798156,-556475
EC00159=-798156,-556475
EC00160=-798156,-556475
EC00161=-798156,-556475
EC00162=-798156,-556475
EC00163=-798156,-556475
EC00164=-798156,-556475
EC00165=-798156,-556475
EC00166=-798156,-556475
EC00167=-798156,-556475
EC00168=-798156,-556475
EC00169=-798156,-556475
EC00170=-798156,-556475
EC00171=-798156,-556475
EC00172=-798156,-556475
EC00173=-798156,-556475
EC00174=-798156,-556475
EC00175=-798156,-556475
EC00176=-798156,-556475
EC00177=-798156,-556475
EC00178=-798156,-556475
EC00179=-798156,-556475
EC00180=-798156,-556475
EC00181=-798156,-556475
EC00182=-798156,-556475
EC00183=-798156,-556475
EC00184=-798156,-556475
EC00185=-798156,-556475
EC00186=-798156,-556475
EC00187=-798156,-556475
EC00188=-798156,-556475
EC00189=-798156,-556475
EC00190=-798156,-556475
EC00191=-798156,-556475
EC00192=-798156,-556475
EC00193=-798156,-556475
EC00194=-798156,-556475
EC00195=-798156,-556475
EC00196=-798156,-556475
EC00197=-798156,-556475
EC00198=-798156,-556475
EC00199=-798156,-556475
EC00200=-798156,-556475
EC00201=-798156,-556475
EC00202=-798156,-556475
EC00203=-798156,-556475
EC00204=-798156,-556475
EC00205=-798156,-556475
EC00206=-798156,-556475
EC00207=-798156,-556475
EC00208=-798156,-556475
EC00209=-798156,-556475
EC00210=-798156,-556475
EC00211=-798156,-556475
EC00212=-798156,-556475
EC00213=-798156,-556475
EC00214=-798156,-556475
EC00215=-798156,-556475
EC00216=-798156,-556475
EC00217=-798156,-556475
EC00218=-798156,-556475
EC00219=-798156,-556475
EC00220=-798156,-556475
EC00221=-798156,-556475
EC00222=-798156,-556475
EC00223=-798156,-556475
EC00224=-798156,-556475
EC00225=-798156,-556475
EC00226=-798156,-556475
EC00227=-798156,-556475
EC00228=-798156,-556475
EC00229=-798156,-556475
EC00230=-798156,-556475
EC00231=-798156,-556475
EC00232=-798156,-556475
EC00233=-798156,-556475
EC00234=-798156,-556475
EC00235=-798153,-556475
EC00236=-798156,-556475
EC00237=-798156,-556475
EC00238=-798156,-556475
EC00239=-798156,-556475
EC00240=-798156,-556475
EC00241=-798156,-556475
EC00242=-798156,-556475
EC00243=-798156,-556475
EC00244=-798156,-556475
EC00245=-798156,-556475
EC00246=-798156,-556475
EC00247=-798155,-556476
EC00248=-798155,-556476
EC00249=-798155,-556476
EC00250=-798155,-556475
EC00251=-798155,-556475
EC00252=-798156,-556475
EC00253=-798156,-556475
EC00254=-798156,-556475
EC00255=-798156,-556475
EC00256=-798156,-556475
EC00257=-798156,-556475
EC00258=-798156,-556475
EC00259=-798156,-556475
EC00260=-798156,-556475
EC00261=-798156,-556475
EC00262=-798156,-556475
EC00263=-798156,-556475
EC00264=-798156,-556475
EC00265=-798156,-556475
EC00266=-798156,-556475
EC00267=-798156,-556475
EC00268=-798156,-556475
EC00269=-798156,-556475
EC00270=-798156,-556475
EC00271=-798156,-556475
EC00272=-798156,-556475
EC00273=-798156,-556475
EC00274=-798156,-556475
EC00275=-798156,-556475
EC00276=-798156,-556475
EC00277=-798156,-556475
EC00278=-798156,-556475
EC00279=-798156,-556475
EC00280=-798156,-556475
EC00281=-798156,-556475
EC00282=-798156,-556475
EC00283=-798156,-556475
EC00284=-798156,-556475
EC00285=-798156,-556475
EC00286=-798156,-556475
EC00287=-798156,-556475
EC00288=-798156,-556475
EC00289=-798156,-556475
EC00290=-798156,-556475
EC00291=-798156,-556475
EC00292=-798156,-556475
EC00293=-798156,-556475
EC00294=-798156,-556475
EC00295=-798156,-556475
EC00296=-798156,-556475
EC00297=-798156,-556475
EC00298=-798156,-556475
EC00299=-798156,-556475
EC00300=-798155,-556475
EC00301=-798156,-556475
EC00302=-798156,-556475
EC00303=-798156,-556475
EC00304=-798156,-556475
EC00305=-798156,-556475
EC00306=-798156,-556475
EC00307=-798156,-556475
EC00308=-798156,-556475
EC00309=-798156,-556475
EC00310=-798156,-556475
EC00311=-798156,-556475
EC00312=-798156,-556475
EC00313=-798156,-556475
EC00314=-798156,-556475
EC00315=-798156,-556475
EC00316=-798156,-556475
EC00317=-798156,-556475
EC00318=-798156,-556475
EC00319=-798156,-556475
EC00320=-798156,-556475
EC00321=-798156,-556475
EC00322=-798156,-556475
EC00323=-798156,-556475
EC00324=-798156,-556475
EC00325=-798156,-556475
EC00326=-798156,-556475
EC00327=-798156,-556475
EC00328=-798156,-556475
EC00329=-798156,-556475
EC00330=-798156,-556475
EC00331=-798156,-556475
EC00332=-798156,-556475
EC00333=-798156,-556475
EC00334=-798156,-556475
EC00335=-798156,-556475
EC00336=-798156,-556475
EC00337=-798156,-556475
EC00338=-798156,-556475
EC00339=-798156,-556475
EC00340=-798154,-556475
EC00341=-798154,-556475
EC00342=-798154,-556475
EC00343=-798156,-556475
EC00344=-798156,-556475
EC00345=-798156,-556475
EC00346=-798156,-556475
///POSTYPE BASE
///RECTAN
///RCONF 0,0,0,0,0,0,0,0,0,0,0,0,0,0,0,0,0,0,0,0,0,0,0,0
P00006=0.222,-3.123,-1.508,0.0000,0.0000,0.0000
P00021=-0.225,-6.128,-0.405,0.0000,0.0000,0.0000
P00022=0.222,-3.123,-1.508,0.0000,0.0000,0.0000
P00023=0.143,-0.036,0.682,0.0000,0.0000,0.0000
P00024=0.145,-0.552,1.326,0.0000,0.0000,0.0000
P00025=-2.003,0.006,0.728,0.0000,0.0000,0.0000
P00031=1.853,-0.001,-1.549,0.0000,0.0000,0.0000
P00032=1.957,0.503,-7.217,0.0000,0.0000,0.0000
///RCONF 0,0,0,0,1,0,0,0,0,0,0,0,0,0,0,0,0,0,0,0,0,0,0,0
P00033=-0.123,0.612,-5.012,0.0000,0.0000,0.0000
///RCONF 0,0,0,0,0,0,0,0,0,0,0,0,0,0,0,0,0,0,0,0,0,0,0,0
P00034=-0.304,0.773,-2.693,0.0000,0.0000,0.0000
P00035=2.817,0.591,-1.622,0.0000,0.0000,0.0000
P00036=-1.108,-0.829,1.850,0.0000,0.0000,0.0000
P00037=0.023,0.937,-2.677,0.0000,0.0000,0.0000
P00038=0.158,-1.133,-1.952,0.0000,0.0000,0.0000
P00039=0.012,-3.081,-0.106,0.0000,0.0000,0.0000
P00040=-0.030,9.648,2.467,0.0000,0.0000,0.0000
//INST
///DATE 2024/11/04 15:01
///ATTR SC,RW
///GROUP1 RB1,BS1
///GROUP2 ST1
NOP
'X2_27-28(-50,-90)
'spoiny do polaczenia
MOVJ C00000 BC00000 VJ=100.00  +MOVJ EC00000 VJ=100.00
MOVJ C00001 BC00001 VJ=100.00  +MOVJ EC00001 VJ=100.00
'Path S4320
SSFTOF
SFTOF3D
MOVJ C00002 BC00002 VJ=100.00  +MOVJ EC00002 VJ=100.00
MOVL C00003 BC00003 V=800.0  +MOVJ EC00003 VJ=100.00
SMOVL C00004 BC00004 V=166.7  +MOVJ EC00004
SREFP 3 C00005 BC00005  +REFP EC00005
CALL JOB:SEARCH-R1-S13D
SET P033 P006
SFTON3D P033
SMOVL C00006 BC00006 V=166.7  +MOVJ EC00006
SREFP 3 C00007 BC00007  +REFP EC00007
CALL JOB:SEARCH-R1-S13D
SET P033 P006
SFTON3D P033
SMOVL C00008 BC00008 V=166.7  +MOVJ EC00008
SMOVL C00009 BC00009 V=166.7  +MOVJ EC00009
SREFP 3 C00010 BC00010  +REFP EC00010
CALL JOB:SEARCH-R1-S13D
SET P033 P006
SFTON3D P033
SMOVL C00011 BC00011 V=166.7  +MOVJ EC00011
MOVL C00012 BC00012 V=800.0  +MOVJ EC00012 VJ=100.00
MOVL C00013 BC00013 V=1000.0  +MOVJ EC00013 VJ=100.00
'EndPath S4320
'Path S4321
SFTOF3D
MOVJ C00014 BC00014 VJ=100.00  +MOVJ EC00014 VJ=100.00
MOVL C00015 BC00015 V=800.0  +MOVJ EC00015 VJ=100.00
SMOVL C00016 BC00016 V=166.7  +MOVJ EC00016
SREFP 3 C00017 BC00017  +REFP EC00017
CALL JOB:SEARCH-R1-S13D
SET P034 P006
SFTON3D P034
SMOVL C00018 BC00018 V=166.7  +MOVJ EC00018
SREFP 3 C00019 BC00019  +REFP EC00019
CALL JOB:SEARCH-R1-S13D
SET P034 P006
SFTON3D P034
SMOVL C00020 BC00020 V=166.7  +MOVJ EC00020
SMOVL C00021 BC00021 V=250.0  +MOVJ EC00021
SMOVL C00022 BC00022 V=166.7  +MOVJ EC00022
SREFP 3 C00023 BC00023  +REFP EC00023
CALL JOB:SEARCH-R1-S13D
SET P034 P006
SFTON3D P034
SMOVL C00024 BC00024 V=166.7  +MOVJ EC00024
MOVL C00025 BC00025 V=1000.0  +MOVJ EC00025 VJ=100.00
'EndPath S4321
'Path S4322
SFTOF3D
MOVJ C00026 BC00026 VJ=100.00  +MOVJ EC00026 VJ=100.00
MOVL C00027 BC00027 V=800.0  +MOVJ EC00027 VJ=100.00
SMOVL C00028 BC00028 V=166.7  +MOVJ EC00028
SREFP 3 C00029 BC00029  +REFP EC00029
CALL JOB:SEARCH-R1-S13D
SET P035 P006
SFTON3D P035
SMOVL C00030 BC00030 V=166.7  +MOVJ EC00030
SREFP 3 C00031 BC00031  +REFP EC00031
CALL JOB:SEARCH-R1-S13D
SET P035 P006
SFTON3D P035
SMOVL C00032 BC00032 V=166.7  +MOVJ EC00032
SMOVL C00033 BC00033 V=250.0  +MOVJ EC00033
SREFP 3 C00034 BC00034  +REFP EC00034
CALL JOB:SEARCH-R1-S13D
SET P035 P006
SFTON3D P035
SMOVL C00035 BC00035 V=250.0  +MOVJ EC00035
MOVL C00036 BC00036 V=1000.0  +MOVJ EC00036 VJ=100.00
'EndPath S4322
'Path S4323
SFTOF3D
MOVJ C00037 BC00037 VJ=100.00  +MOVJ EC00037 VJ=100.00
MOVL C00038 BC00038 V=800.0  +MOVJ EC00038 VJ=100.00
SMOVL C00039 BC00039 V=166.7  +MOVJ EC00039
SREFP 3 C00040 BC00040  +REFP EC00040
CALL JOB:SEARCH-R1-S13D
SET P036 P006
SFTON3D P036
SMOVL C00041 BC00041 V=166.7  +MOVJ EC00041
SREFP 3 C00042 BC00042  +REFP EC00042
CALL JOB:SEARCH-R1-S13D
SET P036 P006
SFTON3D P036
SMOVL C00043 BC00043 V=166.7  +MOVJ EC00043
SMOVL C00044 BC00044 V=250.0  +MOVJ EC00044
SREFP 3 C00045 BC00045  +REFP EC00045
CALL JOB:SEARCH-R1-S13D
SET P036 P006
SFTON3D P036
SMOVL C00046 BC00046 V=250.0  +MOVJ EC00046
MOVL C00047 BC00047 V=1000.0  +MOVJ EC00047 VJ=100.00
'EndPath S4323
'
MOVJ C00048 BC00048 VJ=100.00  +MOVJ EC00048 VJ=100.00
'Path S4328
SFTOF3D
MOVJ C00049 BC00049 VJ=100.00  +MOVJ EC00049 VJ=100.00
MOVL C00050 BC00050 V=800.0  +MOVJ EC00050 VJ=100.00
SMOVL C00051 BC00051 V=166.7  +MOVJ EC00051
SREFP 3 C00052 BC00052  +REFP EC00052
CALL JOB:SEARCH-R1-S13D
SET P040 P006
SFTON3D P040
SMOVL C00053 BC00053 V=166.7  +MOVJ EC00053
SREFP 3 C00054 BC00054  +REFP EC00054
CALL JOB:SEARCH-R1-S13D
SET P040 P006
SFTON3D P040
SMOVL C00055 BC00055 V=166.7  +MOVJ EC00055
SMOVL C00056 BC00056 V=250.0  +MOVJ EC00056
SREFP 3 C00057 BC00057  +REFP EC00057
CALL JOB:SEARCH-R1-S13D
SET P040 P006
SFTON3D P040
SMOVL C00058 BC00058 V=250.0  +MOVJ EC00058
MOVL C00059 BC00059 V=1000.0  +MOVJ EC00059 VJ=100.00
'EndPath S4328
'Path S4327
SFTOF3D
MOVJ C00060 BC00060 VJ=100.00  +MOVJ EC00060 VJ=100.00
MOVL C00061 BC00061 V=800.0  +MOVJ EC00061 VJ=100.00
SMOVL C00062 BC00062 V=166.7  +MOVJ EC00062
SREFP 3 C00063 BC00063  +REFP EC00063
CALL JOB:SEARCH-R1-S13D
SET P039 P006
SFTON3D P039
SMOVL C00064 BC00064 V=166.7  +MOVJ EC00064
SREFP 3 C00065 BC00065  +REFP EC00065
CALL JOB:SEARCH-R1-S13D
SET P039 P006
SFTON3D P039
SMOVL C00066 BC00066 V=166.7  +MOVJ EC00066
SMOVL C00067 BC00067 V=250.0  +MOVJ EC00067
SREFP 3 C00068 BC00068  +REFP EC00068
CALL JOB:SEARCH-R1-S13D
SET P039 P006
SFTON3D P039
SMOVL C00069 BC00069 V=250.0  +MOVJ EC00069
MOVL C00070 BC00070 V=1000.0  +MOVJ EC00070 VJ=100.00
'EndPath S4327
'Path S4325
SFTOF3D
MOVJ C00071 BC00071 VJ=100.00  +MOVJ EC00071 VJ=100.00
MOVL C00072 BC00072 V=666.7  +MOVJ EC00072 VJ=100.00
SMOVL C00073 BC00073 V=166.7  +MOVJ EC00073
SREFP 3 C00074 BC00074  +REFP EC00074
CALL JOB:SEARCH-R1-S13D
SET P038 P006
SFTON3D P038
SMOVL C00075 BC00075 V=166.7  +MOVJ EC00075
SREFP 3 C00076 BC00076  +REFP EC00076
CALL JOB:SEARCH-R1-S13D
SET P038 P006
SFTON3D P038
SMOVL C00077 BC00077 V=166.7  +MOVJ EC00077
SMOVL C00078 BC00078 V=166.7  +MOVJ EC00078
SMOVL C00079 BC00079 V=166.7  +MOVJ EC00079
SREFP 3 C00080 BC00080  +REFP EC00080
CALL JOB:SEARCH-R1-S13D
SET P038 P006
SFTON3D P038
SMOVL C00081 BC00081 V=166.7  +MOVJ EC00081
MOVL C00082 BC00082 V=1000.0  +MOVJ EC00082 VJ=100.00
'EndPath S4325
'Path S4324
SFTOF3D
MOVJ C00083 BC00083 VJ=100.00  +MOVJ EC00083 VJ=100.00
MOVL C00084 BC00084 V=666.7  +MOVJ EC00084 VJ=100.00
SMOVL C00085 BC00085 V=166.7  +MOVJ EC00085
SREFP 3 C00086 BC00086  +REFP EC00086
CALL JOB:SEARCH-R1-S13D
SET P037 P006
SFTON3D P037
SMOVL C00087 BC00087 V=166.7  +MOVJ EC00087
SREFP 3 C00088 BC00088  +REFP EC00088
CALL JOB:SEARCH-R1-S13D
SET P037 P006
SFTON3D P037
SMOVL C00089 BC00089 V=166.7  +MOVJ EC00089
SMOVL C00090 BC00090 V=250.0  +MOVJ EC00090
SREFP 3 C00091 BC00091  +REFP EC00091
CALL JOB:SEARCH-R1-S13D
SET P037 P006
SFTON3D P037
SMOVL C00092 BC00092 V=250.0  +MOVJ EC00092
MOVL C00093 BC00093 V=1000.0  +MOVJ EC00093 VJ=100.00
'EndPath S4324
'Path W4326
SFTOF3D
SFTON3D P037
MOVJ C00094 BC00094 VJ=100.00  +MOVJ EC00094 VJ=100.00
SMOVL C00095 BC00095 V=800.0  +MOVJ EC00095
SMOVL C00096 BC00096 V=150.0 PL=0  +MOVJ EC00096
MACRO1 MJ#(0) ARGF9
ARCON
SMOVL C00097 BC00097 V=10.0  +MOVJ EC00097
SMOVL C00098 BC00098 V=10.0  +MOVJ EC00098
ARCON
SFTON3D P038
SMOVL C00099 BC00099 V=10.0  +MOVJ EC00099
SMOVL C00100 BC00100 V=10.0  +MOVJ EC00100
SMOVL C00101 BC00101 V=10.0  +MOVJ EC00101
ARCON
SMOVL C00102 BC00102 V=10.0  +MOVJ EC00102
SMOVL C00103 BC00103 V=11.7  +MOVJ EC00103
ARCOF
SMOVL C00104 BC00104 V=800.0  +MOVJ EC00104
SMOVL C00105 BC00105 V=1000.0  +MOVJ EC00105
SFTOF3D
'EndPath W4326
MOVJ C00106 BC00106 VJ=100.00  +MOVJ EC00106 VJ=100.00
'Path W4329
SFTOF3D
SFTON3D P040
MOVJ C00107 BC00107 VJ=100.00  +MOVJ EC00107 VJ=100.00
SMOVL C00108 BC00108 V=800.0  +MOVJ EC00108
SMOVL C00109 BC00109 V=150.0 PL=0  +MOVJ EC00109
ARCON
SMOVL C00110 BC00110 V=10.0  +MOVJ EC00110
SMOVL C00111 BC00111 V=10.0  +MOVJ EC00111
SMOVL C00112 BC00112 V=10.0  +MOVJ EC00112
SMOVL C00113 BC00113 V=10.0  +MOVJ EC00113
SFTON3D P039
SMOVL C00114 BC00114 V=8.3  +MOVJ EC00114
SMOVL C00115 BC00115 V=8.3  +MOVJ EC00115
SMOVL C00116 BC00116 V=8.3  +MOVJ EC00116
ARCOF
SMOVL C00117 BC00117 V=800.0  +MOVJ EC00117
SMOVL C00118 BC00118 V=1000.0  +MOVJ EC00118
SFTOF3D
'EndPath W4329
MOVJ C00119 BC00119 VJ=100.00  +MOVJ EC00119 VJ=100.00
'Path W4330
SFTOF3D
SFTON3D P033
MOVJ C00120 BC00120 VJ=100.00  +MOVJ EC00120 VJ=100.00
SMOVL C00121 BC00121 V=800.0  +MOVJ EC00121
SMOVL C00122 BC00122 V=150.0 PL=0  +MOVJ EC00122
ARCON
SMOVL C00123 BC00123 V=10.0  +MOVJ EC00123
SMOVL C00124 BC00124 V=10.0  +MOVJ EC00124
SFTON3D P034
SMOVL C00125 BC00125 V=10.0  +MOVJ EC00125
SMOVL C00126 BC00126 V=11.7  +MOVJ EC00126
SMOVL C00127 BC00127 V=11.7  +MOVJ EC00127
SMOVL C00128 BC00128 V=11.7  +MOVJ EC00128
ARCOF
SMOVL C00129 BC00129 V=800.0  +MOVJ EC00129
SMOVL C00130 BC00130 V=1000.0  +MOVJ EC00130
SFTOF3D
'EndPath W4330
MOVJ C00131 BC00131 VJ=100.00  +MOVJ EC00131 VJ=100.00
'Path W3572
SFTOF3D
SFTON3D P036
MOVJ C00132 BC00132 VJ=100.00  +MOVJ EC00132 VJ=100.00
SMOVL C00133 BC00133 V=800.0  +MOVJ EC00133
SMOVL C00134 BC00134 V=150.0 PL=0  +MOVJ EC00134
ARCON
SMOVL C00135 BC00135 V=10.0  +MOVJ EC00135
SMOVL C00136 BC00136 V=10.0  +MOVJ EC00136
SMOVL C00137 BC00137 V=10.0  +MOVJ EC00137
SMOVL C00138 BC00138 V=10.0  +MOVJ EC00138
SFTON3D P035
SMOVL C00139 BC00139 V=8.3  +MOVJ EC00139
SMOVL C00140 BC00140 V=8.3  +MOVJ EC00140
SMOVL C00141 BC00141 V=8.3  +MOVJ EC00141
ARCOF
SMOVL C00142 BC00142 V=800.0  +MOVJ EC00142
SMOVL C00143 BC00143 V=1000.0  +MOVJ EC00143
SFTOF3D
'EndPath W3572
MOVJ C00144 BC00144 VJ=100.00  +MOVJ EC00144 VJ=100.00
'
CALL JOB:CLEAN-R1_KM_NEW
MOVJ C00145 BC00145 VJ=100.00  +MOVJ EC00145 VJ=100.00
MOVJ C00146 BC00146 VJ=100.00  +MOVJ EC00146 VJ=100.00
MOVJ C00147 BC00147 VJ=100.00  +MOVJ EC00147 VJ=100.00
COMM PAUSE
COMM MOVJ C00148 BC00148 VJ=100.00  +MOVJ EC00148 VJ=100.00
COMM MOVL C00149 BC00149 V=800.0  +MOVJ EC00149 VJ=100.00
COMM SMOVL C00150 BC00150 V=166.7  +MOVJ EC00150
COMM SREFP 3 C00151 BC00151  +REFP EC00151
COMM CALL JOB:SEARCH-R1-S13D
COMM SET P021 P006
COMM SFTON3D P021
COMM SMOVL C00152 BC00152 V=166.7  +MOVJ EC00152
COMM SREFP 3 C00153 BC00153  +REFP EC00153
COMM CALL JOB:SEARCH-R1-S13D
COMM SET P021 P006
COMM SFTON3D P021
COMM SMOVL C00154 BC00154 V=166.7  +MOVJ EC00154
COMM SMOVL C00155 BC00155 V=250.0  +MOVJ EC00155
COMM SMOVL C00156 BC00156 V=166.7  +MOVJ EC00156
COMM SREFP 3 C00157 BC00157  +REFP EC00157
COMM CALL JOB:SEARCH-R1-S13D
COMM SET P021 P006
COMM SFTON3D P021
COMM SMOVL C00158 BC00158 V=166.7  +MOVJ EC00158
COMM MOVL C00159 BC00159 V=1000.0  +MOVJ EC00159 VJ=100.00
COMM 'EndPath S4299
COMM 'Path S4300
COMM SFTOF3D
COMM MOVJ C00160 BC00160 VJ=100.00  +MOVJ EC00160 VJ=100.00
MOVL C00161 BC00161 V=800.0  +MOVJ EC00161 VJ=100.00
SMOVL C00162 BC00162 V=166.7  +MOVJ EC00162
SREFP 3 C00163 BC00163  +REFP EC00163
CALL JOB:SEARCH-R1-S13D
SET P022 P006
SFTON3D P022
SMOVL C00164 BC00164 V=166.7  +MOVJ EC00164
SMOVL C00165 BC00165 V=166.7  +MOVJ EC00165
SREFP 3 C00166 BC00166  +REFP EC00166
CALL JOB:SEARCH-R1-S13D
SET P022 P006
SFTON3D P022
SMOVL C00167 BC00167 V=166.7  +MOVJ EC00167
SMOVL C00168 BC00168 V=250.0  +MOVJ EC00168
SMOVL C00169 BC00169 V=166.7  +MOVJ EC00169
SREFP 3 C00170 BC00170  +REFP EC00170
CALL JOB:SEARCH-R1-S13D
SET P022 P006
SFTON3D P022
SMOVL C00171 BC00171 V=166.7  +MOVJ EC00171
MOVL C00172 BC00172 V=1000.0  +MOVJ EC00172 VJ=100.00
'EndPath S4300
'Path S4301
SFTOF3D
MOVJ C00173 BC00173 VJ=100.00  +MOVJ EC00173 VJ=100.00
MOVL C00174 BC00174 V=800.0  +MOVJ EC00174 VJ=100.00
SMOVL C00175 BC00175 V=166.7  +MOVJ EC00175
SREFP 3 C00176 BC00176  +REFP EC00176
CALL JOB:SEARCH-R1-S13D
SET P023 P006
SFTON3D P023
SMOVL C00177 BC00177 V=166.7  +MOVJ EC00177
SREFP 3 C00178 BC00178  +REFP EC00178
CALL JOB:SEARCH-R1-S13D
SET P023 P006
SFTON3D P023
SMOVL C00179 BC00179 V=166.7  +MOVJ EC00179
MOVL C00180 BC00180 V=1000.0  +MOVJ EC00180 VJ=100.00
'EndPath S4301
'Path S4302
SFTOF3D
MOVJ C00181 BC00181 VJ=100.00  +MOVJ EC00181 VJ=100.00
MOVL C00182 BC00182 V=800.0  +MOVJ EC00182 VJ=100.00
SMOVL C00183 BC00183 V=166.7  +MOVJ EC00183
SREFP 3 C00184 BC00184  +REFP EC00184
CALL JOB:SEARCH-R1-S13D
SET P024 P006
SFTON3D P024
SMOVL C00185 BC00185 V=166.7  +MOVJ EC00185
SREFP 3 C00186 BC00186  +REFP EC00186
CALL JOB:SEARCH-R1-S13D
SET P024 P006
SFTON3D P024
SMOVL C00187 BC00187 V=166.7  +MOVJ EC00187
MOVL C00188 BC00188 V=1000.0  +MOVJ EC00188 VJ=100.00
'EndPath S4302
'Path S4303
SFTOF3D
MOVJ C00189 BC00189 VJ=100.00  +MOVJ EC00189 VJ=100.00
MOVL C00190 BC00190 V=800.0  +MOVJ EC00190 VJ=100.00
SMOVL C00191 BC00191 V=166.7  +MOVJ EC00191
SREFP 3 C00192 BC00192  +REFP EC00192
CALL JOB:SEARCH-R1-S13D
SET P025 P006
SFTON3D P025
SMOVL C00193 BC00193 V=166.7  +MOVJ EC00193
SREFP 3 C00194 BC00194  +REFP EC00194
CALL JOB:SEARCH-R1-S13D
SET P025 P006
SFTON3D P025
SMOVL C00195 BC00195 V=166.7  +MOVJ EC00195
MOVL C00196 BC00196 V=1000.0  +MOVJ EC00196 VJ=100.00
'EndPath S4303
'Path S4313
SFTOF3D
MOVJ C00197 BC00197 VJ=100.00  +MOVJ EC00197 VJ=100.00
MOVL C00198 BC00198 V=800.0  +MOVJ EC00198 VJ=100.00
SMOVL C00199 BC00199 V=166.7  +MOVJ EC00199
SREFP 3 C00200 BC00200  +REFP EC00200
CALL JOB:SEARCH-R1-S13D
SET P032 P006
SFTON3D P032
SMOVL C00201 BC00201 V=166.7  +MOVJ EC00201
SREFP 3 C00202 BC00202  +REFP EC00202
CALL JOB:SEARCH-R1-S13D
SET P032 P006
SFTON3D P032
SMOVL C00203 BC00203 V=166.7  +MOVJ EC00203
SMOVL C00204 BC00204 V=250.0  +MOVJ EC00204
SMOVL C00205 BC00205 V=166.7  +MOVJ EC00205
SREFP 3 C00206 BC00206  +REFP EC00206
CALL JOB:SEARCH-R1-S13D
SET P032 P006
SFTON3D P032
SMOVL C00207 BC00207 V=166.7  +MOVJ EC00207
MOVL C00208 BC00208 V=1000.0  +MOVJ EC00208 VJ=100.00
'EndPath S4313
'Path S4312
SFTOF3D
MOVJ C00209 BC00209 VJ=100.00  +MOVJ EC00209 VJ=100.00
COMM PAUSE
COMM MOVL C00210 BC00210 V=800.0  +MOVJ EC00210 VJ=100.00
COMM SMOVL C00211 BC00211 V=166.7  +MOVJ EC00211
COMM SREFP 3 C00212 BC00212  +REFP EC00212
COMM CALL JOB:SEARCH-R1-S13D
COMM SET P031 P006
COMM SFTON3D P031
COMM SMOVL C00213 BC00213 V=166.7  +MOVJ EC00213
COMM SREFP 3 C00214 BC00214  +REFP EC00214
COMM CALL JOB:SEARCH-R1-S13D
COMM SET P031 P006
COMM SFTON3D P031
COMM SMOVL C00215 BC00215 V=166.7  +MOVJ EC00215
COMM SMOVL C00216 BC00216 V=250.0  +MOVJ EC00216
COMM SMOVL C00217 BC00217 V=166.7  +MOVJ EC00217
COMM SREFP 3 C00218 BC00218  +REFP EC00218
COMM CALL JOB:SEARCH-R1-S13D
COMM SET P031 P006
COMM SFTON3D P031
COMM SMOVL C00219 BC00219 V=250.0  +MOVJ EC00219
COMM MOVL C00220 BC00220 V=1000.0  +MOVJ EC00220 VJ=100.00
COMM 'EndPath S4312
COMM 'Path W4314
COMM SFTOF3D
COMM SFTON3D P031
COMM MOVJ C00221 BC00221 VJ=100.00  +MOVJ EC00221 VJ=100.00
COMM SMOVL C00222 BC00222 V=800.0  +MOVJ EC00222
COMM SMOVL C00223 BC00223 V=150.0 PL=0  +MOVJ EC00223
COMM MACRO1 MJ#(0) ARGF14
COMM ARCON
COMM SMOVL C00224 BC00224 V=11.7  +MOVJ EC00224
COMM SMOVL C00225 BC00225 V=11.7  +MOVJ EC00225
COMM ARCON
COMM SMOVL C00226 BC00226 V=11.7  +MOVJ EC00226
COMM ARCOF
COMM SMOVL C00227 BC00227 V=800.0  +MOVJ EC00227
COMM SMOVL C00228 BC00228 V=1000.0  +MOVJ EC00228
COMM SFTOF3D
COMM 'EndPath W4314
COMM 'Path W4315
COMM SFTOF3D
COMM SFTON3D P031
COMM MOVJ C00229 BC00229 VJ=100.00  +MOVJ EC00229 VJ=100.00
COMM SMOVL C00230 BC00230 V=800.0  +MOVJ EC00230
COMM SMOVL C00231 BC00231 V=150.0 PL=0  +MOVJ EC00231
COMM MACRO1 MJ#(0) ARGF6
COMM ARCON
COMM SMOVL C00232 BC00232 V=10.8  +MOVJ EC00232
COMM SMOVL C00233 BC00233 V=10.8  +MOVJ EC00233
COMM SMOVL C00234 BC00234 V=10.0  +MOVJ EC00234
COMM SMOVL C00235 BC00235 V=10.0  +MOVJ EC00235
COMM ARCOF
COMM SMOVL C00236 BC00236 V=800.0  +MOVJ EC00236
COMM SMOVL C00237 BC00237 V=333.3  +MOVJ EC00237
COMM SMOVL C00238 BC00238 V=133.3  +MOVJ EC00238
COMM ARCON
COMM SMOVL C00239 BC00239 V=11.7  +MOVJ EC00239
COMM SMOVL C00240 BC00240 V=11.7  +MOVJ EC00240
COMM ARCOF
COMM SMOVL C00241 BC00241 V=250.0  +MOVJ EC00241
COMM SMOVL C00242 BC00242 V=1000.0  +MOVJ EC00242
COMM SFTOF3D
COMM 'EndPath W4315
MOVJ C00243 BC00243 VJ=100.00  +MOVJ EC00243 VJ=100.00
'
'Path W4316
SFTOF3D
SFTON3D P032
MOVJ C00244 BC00244 VJ=100.00  +MOVJ EC00244 VJ=100.00
SMOVL C00245 BC00245 V=800.0  +MOVJ EC00245
SMOVL C00246 BC00246 V=150.0 PL=0  +MOVJ EC00246
MACRO1 MJ#(0) ARGF21
ARCON
SMOVL C00247 BC00247 V=10.0  +MOVJ EC00247
SMOVL C00248 BC00248 V=10.0  +MOVJ EC00248
SMOVL C00249 BC00249 V=8.3  +MOVJ EC00249
ARCON
SMOVL C00250 BC00250 V=9.2  +MOVJ EC00250
SMOVL C00251 BC00251 V=9.2  +MOVJ EC00251
ARCOF
SMOVL C00252 BC00252 V=800.0  +MOVJ EC00252
SMOVL C00253 BC00253 V=1000.0  +MOVJ EC00253
SFTOF3D
'EndPath W4316
MOVJ C00254 BC00254 VJ=100.00  +MOVJ EC00254 VJ=100.00
MOVJ C00255 BC00255 VJ=100.00  +MOVJ EC00255 VJ=100.00
MOVJ C00256 BC00256 VJ=100.00  +MOVJ EC00256 VJ=100.00
'Path W4317
SFTOF3D
SFTON3D P032
MOVJ C00257 BC00257 VJ=100.00  +MOVJ EC00257 VJ=100.00
SMOVL C00258 BC00258 V=800.0  +MOVJ EC00258
SMOVL C00259 BC00259 V=150.0 PL=0  +MOVJ EC00259
ARCON
SMOVL C00260 BC00260 V=10.0  +MOVJ EC00260
SMOVL C00261 BC00261 V=10.0  +MOVJ EC00261
SMOVL C00262 BC00262 V=10.0  +MOVJ EC00262
ARCON
SMOVL C00263 BC00263 V=10.0  +MOVJ EC00263
ARCOF
SMOVL C00264 BC00264 V=800.0  +MOVJ EC00264
SMOVL C00265 BC00265 V=1000.0  +MOVJ EC00265
SFTOF3D
'EndPath W4317
MOVJ C00266 BC00266 VJ=100.00  +MOVJ EC00266 VJ=100.00
'Path W4318
SFTOF3D
SFTON3D P032
MOVJ C00267 BC00267 VJ=100.00  +MOVJ EC00267 VJ=100.00
SMOVL C00268 BC00268 V=800.0  +MOVJ EC00268
SMOVL C00269 BC00269 V=150.0 PL=0  +MOVJ EC00269
SWVON WEV#(99)
MACRO1 MJ#(0) ARGF9
ARCON
SMOVL C00270 BC00270 V=9.2  +MOVJ EC00270
ARCOF
SWVOF
SMOVL C00271 BC00271 V=33.3  +MOVJ EC00271
TIMER T=2.00
ARCON
TIMER T=0.50
SMOVL C00272 BC00272 V=8.3  +MOVJ EC00272
ARCOF
SMOVL C00273 BC00273 V=800.0  +MOVJ EC00273
SFTOF3D
'EndPath W4318
MOVJ C00274 BC00274 VJ=100.00  +MOVJ EC00274 VJ=100.00
'
'Path W4310
SFTOF3D
SFTON3D P024
MOVJ C00275 BC00275 VJ=100.00  +MOVJ EC00275 VJ=100.00
SMOVL C00276 BC00276 V=800.0  +MOVJ EC00276
SMOVL C00277 BC00277 V=150.0 PL=0  +MOVJ EC00277
MACRO1 MJ#(0) ARGF14
ARCON
SWVON WEV#(22)
SMOVL C00278 BC00278 V=10.0  +MOVJ EC00278
SFTON3D P025
SMOVL C00279 BC00279 V=10.0  +MOVJ EC00279
SMOVL C00280 BC00280 V=10.0  +MOVJ EC00280
ARCOF
SWVOF
SMOVL C00281 BC00281 V=800.0  +MOVJ EC00281
SMOVL C00282 BC00282 V=1000.0  +MOVJ EC00282
SFTOF3D
'EndPath W4310
'Path W4311
SFTOF3D
SFTON3D P024
MOVJ C00283 BC00283 VJ=100.00  +MOVJ EC00283 VJ=100.00
SMOVL C00284 BC00284 V=800.0  +MOVJ EC00284
SMOVL C00285 BC00285 V=150.0 PL=0  +MOVJ EC00285
ARCON
SWVON WEV#(22)
SMOVL C00286 BC00286 V=10.0  +MOVJ EC00286
SFTON3D P023
SMOVL C00287 BC00287 V=10.0  +MOVJ EC00287
SMOVL C00288 BC00288 V=10.0  +MOVJ EC00288
ARCOF
SWVOF
SMOVL C00289 BC00289 V=800.0  +MOVJ EC00289
SMOVL C00290 BC00290 V=1000.0  +MOVJ EC00290
SFTOF3D
'EndPath W4311
'
MOVJ C00291 BC00291 VJ=100.00  +MOVJ EC00291 VJ=100.00
MOVJ C00292 BC00292 VJ=100.00  +MOVJ EC00292 VJ=100.00
MOVJ C00293 BC00293 VJ=100.00  +MOVJ EC00293 VJ=100.00
'Path W4331
SFTOF3D
SFTON3D P022
MOVJ C00294 BC00294 VJ=100.00  +MOVJ EC00294 VJ=100.00
SMOVL C00295 BC00295 V=800.0  +MOVJ EC00295
SMOVL C00296 BC00296 V=150.0 PL=0  +MOVJ EC00296
MACRO1 MJ#(0) ARGF21
ARCON
SMOVL C00297 BC00297 V=9.2  +MOVJ EC00297
SMOVL C00298 BC00298 V=9.2  +MOVJ EC00298
SMOVL C00299 BC00299 V=9.2  +MOVJ EC00299
SMOVL C00300 BC00300 V=9.2  +MOVJ EC00300
ARCOF
SFTOF3D
SMOVL C00301 BC00301 V=800.0  +MOVJ EC00301
SMOVL C00302 BC00302 V=333.3  +MOVJ EC00302
SFTOF3D
'EndPath W4331
MOVJ C00303 BC00303 VJ=100.00  +MOVJ EC00303 VJ=100.00
MOVJ C00304 BC00304 VJ=100.00  +MOVJ EC00304 VJ=100.00
'Path W4306
SFTOF3D
SFTON3D P022
MOVJ C00305 BC00305 VJ=100.00  +MOVJ EC00305 VJ=100.00
SMOVL C00306 BC00306 V=800.0  +MOVJ EC00306
SMOVL C00307 BC00307 V=150.0 PL=0  +MOVJ EC00307
ARCON
SMOVL C00308 BC00308 V=10.0  +MOVJ EC00308
SMOVL C00309 BC00309 V=10.0  +MOVJ EC00309
SMOVL C00310 BC00310 V=10.0  +MOVJ EC00310
ARCOF
SMOVL C00311 BC00311 V=800.0  +MOVJ EC00311
SMOVL C00312 BC00312 V=1000.0  +MOVJ EC00312
SFTOF3D
'EndPath W4306
MOVJ C00313 BC00313 VJ=100.00  +MOVJ EC00313 VJ=100.00
'Path W4332
SFTOF3D
SFTON3D P022
MOVJ C00314 BC00314 VJ=100.00  +MOVJ EC00314 VJ=100.00
SMOVL C00315 BC00315 V=800.0  +MOVJ EC00315
SMOVL C00316 BC00316 V=150.0 PL=0  +MOVJ EC00316
SMOVL C00317 BC00317 V=9.2  +MOVJ EC00317
MACRO1 MJ#(0) ARGF9
ARCON
SWVON WEV#(99)
SMOVL C00318 BC00318 V=9.2  +MOVJ EC00318
ARCOF
SWVOF
SMOVL C00319 BC00319 V=9.2  +MOVJ EC00319
TIMER T=3.00
ARCON
SMOVL C00320 BC00320 V=9.2  +MOVJ EC00320
ARCOF
SMOVL C00321 BC00321 V=800.0  +MOVJ EC00321
SFTOF3D
'EndPath W4332
'
MOVJ C00322 BC00322 VJ=100.00  +MOVJ EC00322 VJ=100.00
COMM PAUSE
COMM 'Path W4304
COMM SFTOF3D
COMM SFTON3D P021
COMM MOVJ C00323 BC00323 VJ=100.00  +MOVJ EC00323 VJ=100.00
COMM SMOVL C00324 BC00324 V=800.0  +MOVJ EC00324
COMM SMOVL C00325 BC00325 V=150.0 PL=0  +MOVJ EC00325
COMM MACRO1 MJ#(0) ARGF14
COMM ARCON
COMM SMOVL C00326 BC00326 V=10.0  +MOVJ EC00326
COMM SMOVL C00327 BC00327 V=10.0  +MOVJ EC00327
COMM SMOVL C00328 BC00328 V=10.0  +MOVJ EC00328
COMM ARCOF
COMM SMOVL C00329 BC00329 V=800.0  +MOVJ EC00329
COMM SMOVL C00330 BC00330 V=1000.0  +MOVJ EC00330
COMM SFTOF3D
COMM 'EndPath W4304
COMM 'Path W4305
COMM SFTOF3D
COMM SFTON3D P021
COMM MOVJ C00331 BC00331 VJ=100.00  +MOVJ EC00331 VJ=100.00
COMM SMOVL C00332 BC00332 V=800.0  +MOVJ EC00332
COMM SMOVL C00333 BC00333 V=150.0 PL=0  +MOVJ EC00333
COMM MACRO1 MJ#(0) ARGF6
COMM ARCON
COMM SMOVL C00334 BC00334 V=10.8  +MOVJ EC00334
COMM SMOVL C00335 BC00335 V=10.8  +MOVJ EC00335
COMM SMOVL C00336 BC00336 V=10.8  +MOVJ EC00336
COMM SMOVL C00337 BC00337 V=11.7  +MOVJ EC00337
COMM ARCOF
COMM SMOVL C00338 BC00338 V=800.0  +MOVJ EC00338
COMM SMOVL C00339 BC00339 V=333.3  +MOVJ EC00339
COMM SMOVL C00340 BC00340 V=333.3  +MOVJ EC00340
COMM ARCON
COMM SMOVL C00341 BC00341 V=11.7  +MOVJ EC00341
COMM ARCOF
COMM SMOVL C00342 BC00342 V=333.3  +MOVJ EC00342
COMM SMOVL C00343 BC00343 V=1000.0  +MOVJ EC00343
COMM SFTOF3D
COMM 'EndPath W4305
MOVJ C00344 BC00344 VJ=100.00  +MOVJ EC00344 VJ=100.00
MOVJ C00345 BC00345 VJ=100.00  +MOVJ EC00345 VJ=100.00
MOVJ C00346 BC00346 VJ=100.00  +MOVJ EC00346 VJ=100.00
END
